TEXTLIST TL_E_CTRL_XPU
  0 = 'XTS_CMD_NULL'
  10 = 'XTS_CMD_INIT'
  30 = 'XTS_IDLE'
   = ''
END_TEXTLIST

(* stored: Version 1.1.0.1, ProductVersion 3.1.4026.13
   TextList TL_E_CTRL_XPU: Id {6df1a2c1-0ad4-45b8-8105-da5e26a7fa0f} *)
